// TIA Portal V17 export
FUNCTION "FC_VFD_CommFault" : Void   // FC, LAD
{ S7_Optimized_Access := 'TRUE' }
// stored: AutoNumber true
   VAR_TEMP   // added for the SCL form of the ladder/FBD networks
      _w1 : Bool;
      _w2 : Bool;
   END_VAR
BEGIN

REGION Network 1: 变频器通讯故障检测
   // 检测变频器通讯失败/成功的上升沿，置位/复位故障标志；若故障标志保持接通3分钟以上则输出通讯故障报警。
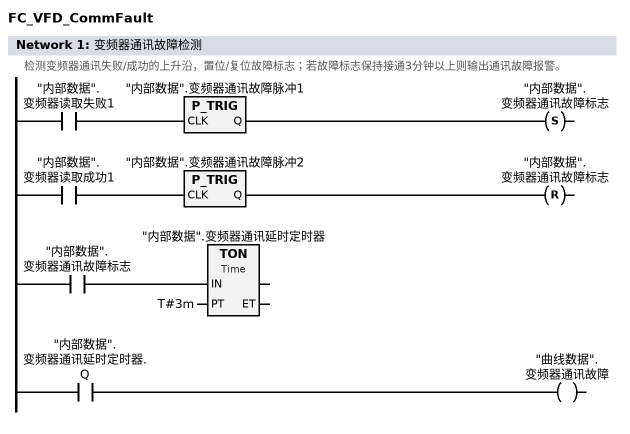
   RUNG wire#powerrail
      Contact( "内部数据".变频器读取失败1 )
      P_Trig( "内部数据".变频器通讯故障脉冲1 )
      S_Coil( "内部数据".变频器通讯故障标志 )
   END_RUNG
   RUNG wire#powerrail
      Contact( "内部数据".变频器读取成功1 )
      P_Trig( "内部数据".变频器通讯故障脉冲2 )
      R_Coil( "内部数据".变频器通讯故障标志 )
   END_RUNG
   RUNG wire#powerrail
      Contact( "内部数据".变频器通讯故障标志 )
      { S7_Templates := "time_type := Time" } "内部数据".变频器通讯延时定时器.TON(pt := T#3m, et =>)
   END_RUNG
   RUNG wire#powerrail
      Contact( "内部数据".变频器通讯延时定时器.Q )
      Coil( "曲线数据".变频器通讯故障 )
   END_RUNG
   // the same network as SCL:
   #_w1 := "内部数据".变频器读取失败1 AND NOT "内部数据".变频器通讯故障脉冲1;   // rising edge
   "内部数据".变频器通讯故障脉冲1 := "内部数据".变频器读取失败1;
   IF #_w1 THEN "内部数据".变频器通讯故障标志 := TRUE; END_IF;
   #_w2 := "内部数据".变频器读取成功1 AND NOT "内部数据".变频器通讯故障脉冲2;   // rising edge
   "内部数据".变频器通讯故障脉冲2 := "内部数据".变频器读取成功1;
   IF #_w2 THEN "内部数据".变频器通讯故障标志 := FALSE; END_IF;
   "内部数据".变频器通讯延时定时器.TON(IN := "内部数据".变频器通讯故障标志, PT := T#3m);
   "曲线数据".变频器通讯故障 := "内部数据".变频器通讯延时定时器.Q;
END_REGION
END_FUNCTION
